# EPICS IOC start-up script: test/startup/st.mcu006-Dbg.iocsh
require EthercatMC,USER

epicsEnvSet("ECM_NUMAXES",   "2")
epicsEnvSet("MOTOR_PORT",    "$(SM_MOTOR_PORT=MCU1)")

epicsEnvSet("IPADDR",        "$(SM_IPADDR=172.30.242.17)")
epicsEnvSet("IPPORT",        "$(SM_IPPORT=5000)")
epicsEnvSet("ASYN_PORT",     "$(SM_ASYN_PORT=MC_CPU1)")
epicsEnvSet("PREFIX",        "$(SM_PREFIX=LabS-MCAG:)")
epicsEnvSet("P",             "$(SM_PREFIX=LabS-MCAG:)")
epicsEnvSet("EGU",           "$(SM_EGU=mm)")
epicsEnvSet("PREC",          "$(SM_PREC=3)")

epicsEnvSet("ECM_OPTIONS",          "")
# Controller
< EthercatMCController.iocsh

# Axis 1
epicsEnvSet("MOTOR_NAME",    "$(SM_MOTOR_NAME=MC-MCU-06:m1)")
epicsEnvSet("AXIS_NO",       "$(SM_AXIS_NO=1)")
epicsEnvSet("DESC",          "$(SM_DESC=Axis)")
epicsEnvSet("AXISCONFIG",    "HomProc=1;HomPos=0;encoder=ADSPORT=501/.ADR.16#3040010,16#80000049,2,2")

< EthercatMCAxis.iocsh
< EthercatMCAxisdebug.iocsh
< EthercatMCAxishome.iocsh
